PROGRAM MAIN
VAR
	
END_VAR

APIs();
Testing();

END_PROGRAM

(* stored: Version 1.1.0.1
   POU MAIN: Id {e6b5e1ee-c466-480b-9668-9427c47f7eda}, SpecialFunc None *)
